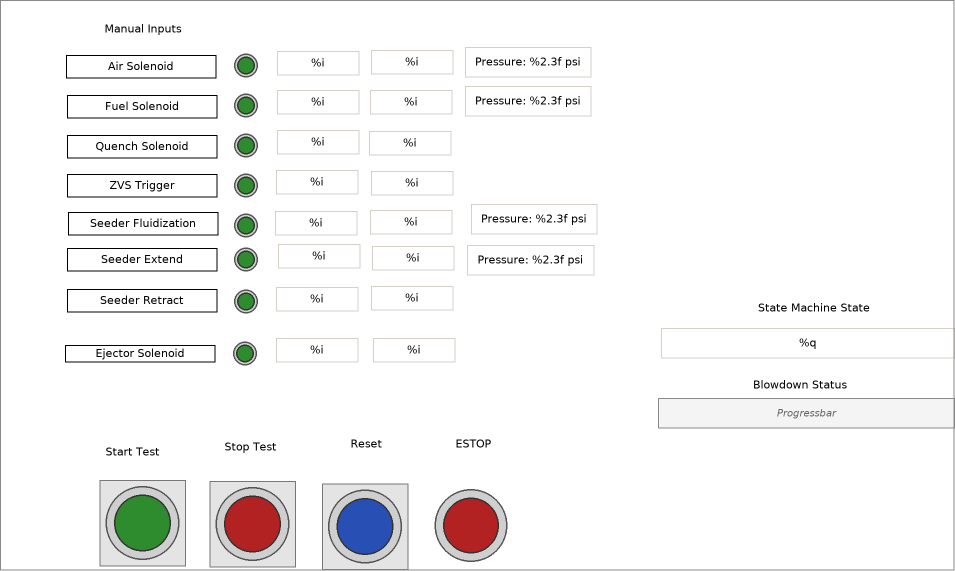
VISUALIZATION Visualization  // 955x571
    RoundedRectangle (66,55 150x23), "Air Solenoid"
        toggle gIO.DO_CombustorAirSolenoid
    RoundedRectangle (67,95 150x23), "Fuel Solenoid"
        toggle gIO.DO_MethaneSolenoid
    RoundedRectangle (67,135 150x23), "Quench Solenoid"
        toggle gIO.DO_WaterQuenchSolenoid
    RoundedRectangle (67,174 150x23), "ZVS Trigger"
        toggle gIO.DO_ZVSIgnite
    RoundedRectangle (68,212 150x23), "Seeder Fluidization"
        toggle gIO.DO_SeederFluidization
    RoundedRectangle (67,248 150x23), "Seeder Extend"
        toggle gIO.DO_SeederExtendSolenoid
    RoundedRectangle (67,289 150x23), "Seeder Retract"
        toggle gIO.DO_SeederRetractSolenoid
    Label (68,14 150x30), "Manual Inputs"
    Lamp1 (232,52 28x27), variable: gIO.DO_CombustorAirSolenoid, style: Lamp-Lamp1-Green
    Lamp1 (232,92 28x27), variable: gIO.DO_MethaneSolenoid, style: Lamp-Lamp1-Green
    Lamp1 (232,132 28x27), variable: gIO.DO_WaterQuenchSolenoid, style: Lamp-Lamp1-Green
    Lamp1 (232,172 28x27), variable: gIO.DO_ZVSIgnite, style: Lamp-Lamp1-Green
    Lamp1 (232,212 28x27), variable: gIO.DO_SeederFluidization, style: Lamp-Lamp1-Green
    Lamp1 (232,246 28x27), variable: gIO.DO_SeederExtendSolenoid, style: Lamp-Lamp1-Green
    Lamp1 (232,288 28x27), variable: gIO.DO_SeederRetractSolenoid, style: Lamp-Lamp1-Green
    PushSwitch (98,480 89x86), variable: MAIN.testFB.command_StartTest, behaviour: TOGGLE, style: Switch-PushSwitch-Green
    PushSwitch (208,481 89x86), tooltip "STOP", variable: MAIN.testFB.command_StopTest, behaviour: TOGGLE, style: Switch-PushSwitch-Red
    Progressbar (658,398 297x30), variable: gHMI.iBlowdownTimeProgress
    Label (725,370 150x30), "Blowdown Status"
    Label (201,432 99x30), "Stop Test"
    Label (83,437 99x30), "Start Test"
    Lamp1 (429,483 84x85), variable: gHMI.bEStopPressed, style: Lamp-Lamp1-Red
    PushSwitch (322,482 86x89), variable: gHMI.bReset, behaviour: TOGGLE, style: Switch-PushSwitch-Blue
    Label (317,429 99x30), "Reset"
    Label (424,429 99x30), "ESTOP"
    Textfield (661,328 294x30), "%q", text variable: gMachine.testCell.state
    Label (739,293 150x30), "State Machine State"
    RoundedRectangle (65,345 150x17), "Ejector Solenoid"
        toggle gIO.DO_EjectorSolenoid
    Lamp1 (231,340 28x27), variable: gIO.DO_EjectorSolenoid, style: Lamp-Lamp1-Green
    Textfield (471,204 126x30), "Pressure: %2.3f psi", text variable: MAIN.monitoredValueUpdate.monitoredValues[5].scaledValue
    Textfield (467,245 127x30), "Pressure: %2.3f psi", text variable: MAIN.monitoredValueUpdate.monitoredValues[6].scaledValue
    Textfield (465,86 126x30), "Pressure: %2.3f psi", text variable: MAIN.monitoredValueUpdate.monitoredValues[2].scaledValue
    Textfield (465,47 126x30), "Pressure: %2.3f psi", text variable: MAIN.monitoredValueUpdate.monitoredValues[1].scaledValue
    Textfield (277,51 82x24), "%i", text variable: gHMI.iAirStartTime
        OnMouseDown: write the text variable via InputWithLimits, min 0, max 50000
    Textfield (371,50 82x24), "%i", text variable: gHMI.iAirStopTime
        OnMouseDown: write the text variable via InputWithLimits, min 0, max 10000
    Textfield (277,90 82x24), "%i", text variable: gHMI.iFuelStartTime
        OnMouseDown: write the text variable via InputWithLimits
    Textfield (370,90 82x24), "%i", text variable: gHMI.iFuelStopTime
        OnMouseDown: write the text variable via InputWithLimits
    Textfield (277,130 82x24), "%i", text variable: gHMI.iWaterQuenchStartTime
        OnMouseDown: write the text variable via InputWithLimits
    Textfield (369,131 82x24), "%i", text variable: gHMI.iWaterQuenchStopTime
        OnMouseDown: write the text variable via InputWithLimits
    Textfield (276,170 82x24), "%i", text variable: gHMI.iZVSStartTime
        OnMouseDown: write the text variable via InputWithLimits, min 0, max 50000
    Textfield (371,171 82x24), "%i", text variable: gHMI.iZVSStopTime
        OnMouseDown: write the text variable via InputWithLimits, min 0, max 50000
    Textfield (370,210 82x24), "%i", text variable: gHMI.iFluidizationStopTime
        OnMouseDown: write the text variable via InputWithLimits, min 0, max 50000
    Textfield (275,211 82x24), "%i", text variable: gHMI.iFluidizationStartTime
        OnMouseDown: write the text variable via InputWithLimits, min 0, max 50000
    Textfield (278,244 82x24), "%i", text variable: gHMI.iSeederExtendStartTime
        OnMouseDown: write the text variable via InputWithLimits, min 0, max 50000
    Textfield (276,287 82x24), "%i", text variable: gHMI.iSeederRetractStartTime
        OnMouseDown: write the text variable via InputWithLimits, min 0, max 50000
    Textfield (371,286 82x24), "%i", text variable: gHMI.iSeederRetractStopTime
        OnMouseDown: write the text variable via VisuDialogs.Keypad, min 0, max 50000
    Textfield (372,246 82x24), "%i", text variable: gHMI.iSeederExtendStopTime
        OnMouseDown: write the text variable via InputWithLimits, min 0, max 50000
    Textfield (276,338 82x24), "%i", text variable: gHMI.iSeederRetractStartTime
        OnMouseDown: write the text variable via InputWithLimits, min 0, max 50000
    Textfield (373,338 82x24), "%i", text variable: gHMI.iSeederRetractStopTime
        OnMouseDown: write the text variable via VisuDialogs.Keypad, min 0, max 50000
END_VISUALIZATION

(* stored: Version 1.1.0.1, ProductVersion 3.1.4024.12
   Visu Visualization: Id {95502d39-bda2-4490-a610-6c7071523a50} *)
